# EPICS IOC start-up script: iocsh/siargo-meter.iocsh
#- ###         MODBUS   siargo   iocsh              ###
#- ####################################################
#- >> Mandatory
#- ASYN_PORT_NAME - MODBUS ASYN <name>
#- PREFIX	  - PV PREFIX
#- MODBUS_ADR	  - Modbus address
#- ASLO		  - linear scale for flow rate (0.001
#- 		    for gauge set for Nm³/h, 0.00006
#-		    for gauge set for SLPM
#- SCALE	  - scale factor for total flow
#  		    (1.0 for gauge set for Nm³,
#-		    0.001 for gauge set for SL)
#-
#- >>> Optional
#- EGU_FR	  - EGU for FlowRt (default Nm³/h)
#- EGU_F	  - EGU Accflow (default Nm³)

#drvModbusAsynConfigure	 'Port name'
#			 'Octet port name'
#			 'Modbus slave address'
#			 'Modbus function code'
#			 'Modbus start address'
#			 'Modbus length'
#			 'Data type'
#			 'Poll time (msec)'
#			 'PLC type'

drvModbusAsynConfigure(RO_DATA_$(ASYN_PORT_NAME)_$(MODBUS_ADR), "$(ASYN_PORT_NAME)", $(MODBUS_ADR), 3, 0x0030, 16, "UINT16", 4000, "siargo")

drvModbusAsynConfigure(WO_DATA_$(ASYN_PORT_NAME)_$(MODBUS_ADR), "$(ASYN_PORT_NAME)", $(MODBUS_ADR), 6, -1, 1, "UINT16", 0, "siargo")

#Load your database defining the EPICS records

dbLoadRecords("siargo.db", "PORT_RO=RO_DATA_$(ASYN_PORT_NAME)_$(MODBUS_ADR),PORT_WO=WO_DATA_$(ASYN_PORT_NAME)_$(MODBUS_ADR),P=$(PREFIX),D=$(DEV_NAME),ASLO=$(ASLO),SCALE=$(SCALE),EGU_FR=$(EGU_FR=Nm³/h),EGU_F=$(EGU_F="Nm³)")
